Staubli VAL3: Control_ListMJ.pgx

public program Control_ListMJ(bool& x_bMJ[], num x_nMoveFirst, num x_nSelectItem)
  local num l_nIndex
  local bool l_bRes
  local string l_sText
begin


//  call Control_ListBas(x_nSelectItem)
//
//
//
//
//  //把列表给画出来
//  for l_nIndex=0 to min(nBottomY-nTopY-1,size(x_bMJ)-x_nMoveFirst)
//
//    setTextMode(0)
//    if x_nMoveFirst+l_nIndex>size(x_bMJ)-1
//      return
//    endIf
//    //MOVEL
//    gotoxy(nTopX+1,nTopY+l_nIndex+1)
//    if !x_bMJ[x_nMoveFirst+l_nIndex]
//      if l_nIndex==x_nSelectItem
//        setTextMode(1)
//      else
//        setTextMode(0)
//      endIf
//      put(left(toString("",x_nMoveFirst+l_nIndex+1)+"       ",4 )+left("MOVEJ             ",24-nBottomX))
//    else
//      //MOVEC
//      if l_nIndex==x_nSelectItem
//        setTextMode(1)
//      else
//        setTextMode(0)
//      endIf
//      put(left(toString("",x_nMoveFirst+l_nIndex+1)+"       ",4 )+left("MOVEL              ",24-nBottomX))
//
//    endIf
//
//  endFor
//

end
